PROGRAM P_InitializeSystem
VAR
END_VAR

END_PROGRAM

(* stored: Version 1.1.0.1, ProductVersion 3.1.4020.12
   POU P_InitializeSystem: Id {9d3c29d9-26b1-439a-a183-dcf5570d24b6}, SpecialFunc None *)
